// TIA Portal V17 export
// export: Created 2023-02-25T15:48:13.2517899Z, ExportSetting WithDefaults, DisplayName Totally Integrated Automation Portal, DisplayVersion V17, DisplayName TIA Portal Openness, DisplayVersion V17, DisplayName TIA Portal Version Control Interface, DisplayVersion V17, DisplayName TIA Portal Test Suite Advanced, DisplayVersion V17, DisplayName STEP 7 Professional, DisplayVersion V17, DisplayName SIMATIC Energy Suite, DisplayVersion V17, DisplayName STEP 7 Safety, DisplayVersion V17, DisplayName WinCC Professional, DisplayVersion V17
FUNCTION_BLOCK "LOG_AutoControle"   // FB5, LAD
TITLE = Auto Controle - Sequential algorithm
{ S7_Optimized_Access := 'TRUE' }
VERSION : 0.1
// stored: AutoNumber true, IsIECCheckEnabled false, IsRetainMemResEnabled false, MemoryReserve 100, SetENOAutomatically false, UDAEnableTagReadback false
   VAR_INPUT
      StartLine : Bool;
      StopLine : Bool;
      AutoMode : Bool;
      SmallPackage : Bool;
      MediumPackage : Bool;
      LargePackage : Bool;
      D3 : Bool;
      D4 : Bool;
      D5 : Bool;
      D6 : Bool;
      FirstScan : Bool;
   END_VAR
   VAR_OUTPUT
      ConveyorsAuto : "stt_Conveyor";
   END_VAR
   VAR
      s1 : Bool;
      s2 : Bool;
      s3 : Bool;
      s4 : Bool;
      s5 : Bool;
      P_D3_1 : Bool;
      P_D3_2 : Bool;
      P_D3_3 : Bool;
      N_D4 : Bool;
      N_D5 : Bool;
      N_D6 : Bool;
   END_VAR
   VAR_TEMP   // added for the SCL form of the ladder/FBD networks
      _w1 : Bool;
   END_VAR
BEGIN

REGION Network 1: Step 3-2
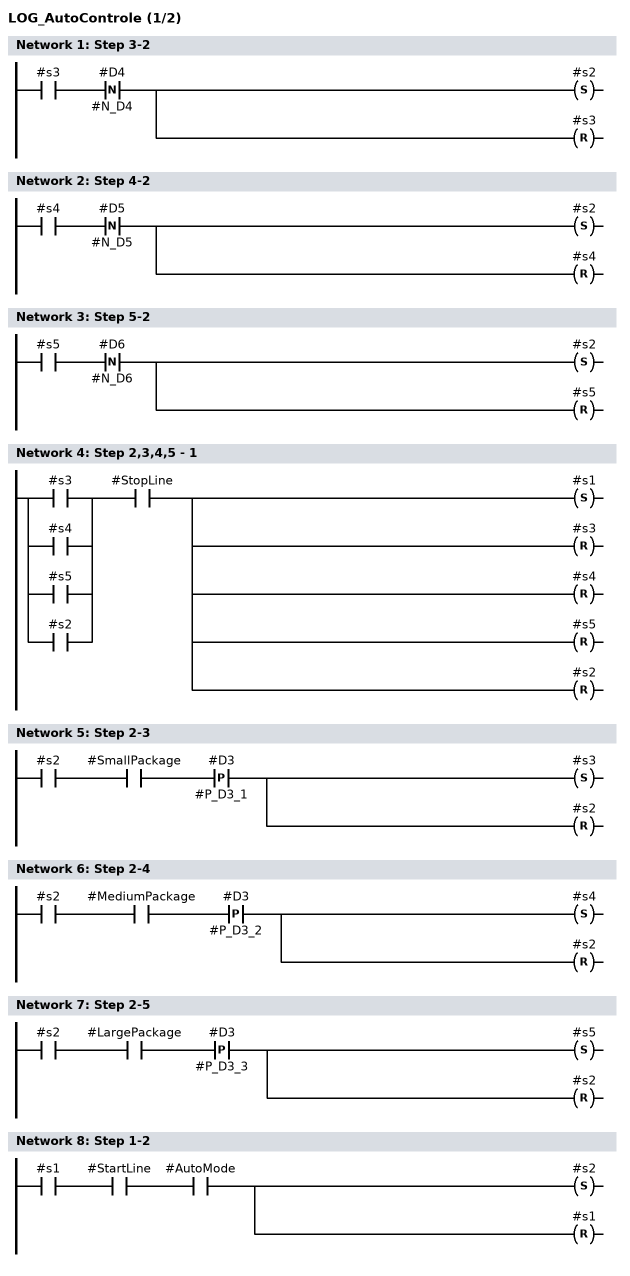
   RUNG wire#powerrail
      Contact( #s3 )
      N_Contact(operand := #D4, bit := #N_D4)
      wire#w1
      S_Coil( #s2 )
   END_RUNG
   RUNG wire#w1
      R_Coil( #s3 )
   END_RUNG
   // the same network as SCL:
   #_w1 := #s3 AND NOT #D4 AND #N_D4;   // falling edge of #D4
   #N_D4 := #D4;
   IF #_w1 THEN
       #s2 := TRUE;
       #s3 := FALSE;
   END_IF;
END_REGION

REGION Network 2: Step 4-2
   RUNG wire#powerrail
      Contact( #s4 )
      N_Contact(operand := #D5, bit := #N_D5)
      wire#w1
      S_Coil( #s2 )
   END_RUNG
   RUNG wire#w1
      R_Coil( #s4 )
   END_RUNG
   // the same network as SCL:
   #_w1 := #s4 AND NOT #D5 AND #N_D5;   // falling edge of #D5
   #N_D5 := #D5;
   IF #_w1 THEN
       #s2 := TRUE;
       #s4 := FALSE;
   END_IF;
END_REGION

REGION Network 3: Step 5-2
   RUNG wire#powerrail
      Contact( #s5 )
      N_Contact(operand := #D6, bit := #N_D6)
      wire#w1
      S_Coil( #s2 )
   END_RUNG
   RUNG wire#w1
      R_Coil( #s5 )
   END_RUNG
   // the same network as SCL:
   #_w1 := #s5 AND NOT #D6 AND #N_D6;   // falling edge of #D6
   #N_D6 := #D6;
   IF #_w1 THEN
       #s2 := TRUE;
       #s5 := FALSE;
   END_IF;
END_REGION

REGION Network 4: Step 2,3,4,5 - 1
   RUNG wire#powerrail
      Contact( #s3 )
      wire#w1
      Contact( #StopLine )
      wire#w2
      S_Coil( #s1 )
   END_RUNG
   RUNG wire#powerrail
      Contact( #s4 )
   END_RUNG wire#w1
   RUNG wire#powerrail
      Contact( #s5 )
   END_RUNG wire#w1
   RUNG wire#powerrail
      Contact( #s2 )
   END_RUNG wire#w1
   RUNG wire#w2
      R_Coil( #s3 )
   END_RUNG
   RUNG wire#w2
      R_Coil( #s4 )
   END_RUNG
   RUNG wire#w2
      R_Coil( #s5 )
   END_RUNG
   RUNG wire#w2
      R_Coil( #s2 )
   END_RUNG
   // the same network as SCL:
   IF (#s3 OR #s4 OR #s5 OR #s2) AND #StopLine THEN #s1 := TRUE; END_IF;
   #_w1 := (#s3 OR #s4 OR #s5 OR #s2) AND #StopLine;
   IF #_w1 THEN
       #s3 := FALSE;
       #s4 := FALSE;
       #s5 := FALSE;
       #s2 := FALSE;
   END_IF;
END_REGION

REGION Network 5: Step 2-3
   RUNG wire#powerrail
      Contact( #s2 )
      Contact( #SmallPackage )
      P_Contact(operand := #D3, bit := #P_D3_1)
      wire#w1
      S_Coil( #s3 )
   END_RUNG
   RUNG wire#w1
      R_Coil( #s2 )
   END_RUNG
   // the same network as SCL:
   #_w1 := #s2 AND #SmallPackage AND #D3 AND NOT #P_D3_1;   // rising edge of #D3
   #P_D3_1 := #D3;
   IF #_w1 THEN
       #s3 := TRUE;
       #s2 := FALSE;
   END_IF;
END_REGION

REGION Network 6: Step 2-4
   RUNG wire#powerrail
      Contact( #s2 )
      Contact( #MediumPackage )
      P_Contact(operand := #D3, bit := #P_D3_2)
      wire#w1
      S_Coil( #s4 )
   END_RUNG
   RUNG wire#w1
      R_Coil( #s2 )
   END_RUNG
   // the same network as SCL:
   #_w1 := #s2 AND #MediumPackage AND #D3 AND NOT #P_D3_2;   // rising edge of #D3
   #P_D3_2 := #D3;
   IF #_w1 THEN
       #s4 := TRUE;
       #s2 := FALSE;
   END_IF;
END_REGION

REGION Network 7: Step 2-5
   RUNG wire#powerrail
      Contact( #s2 )
      Contact( #LargePackage )
      P_Contact(operand := #D3, bit := #P_D3_3)
      wire#w1
      S_Coil( #s5 )
   END_RUNG
   RUNG wire#w1
      R_Coil( #s2 )
   END_RUNG
   // the same network as SCL:
   #_w1 := #s2 AND #LargePackage AND #D3 AND NOT #P_D3_3;   // rising edge of #D3
   #P_D3_3 := #D3;
   IF #_w1 THEN
       #s5 := TRUE;
       #s2 := FALSE;
   END_IF;
END_REGION

REGION Network 8: Step 1-2
   RUNG wire#powerrail
      Contact( #s1 )
      Contact( #StartLine )
      Contact( #AutoMode )
      wire#w1
      S_Coil( #s2 )
   END_RUNG
   RUNG wire#w1
      R_Coil( #s1 )
   END_RUNG
   // the same network as SCL:
   IF #s1 AND #StartLine AND #AutoMode THEN
       #s2 := TRUE;
       #s1 := FALSE;
   END_IF;
END_REGION

REGION Network 9: Step 2,3,4,5 Output
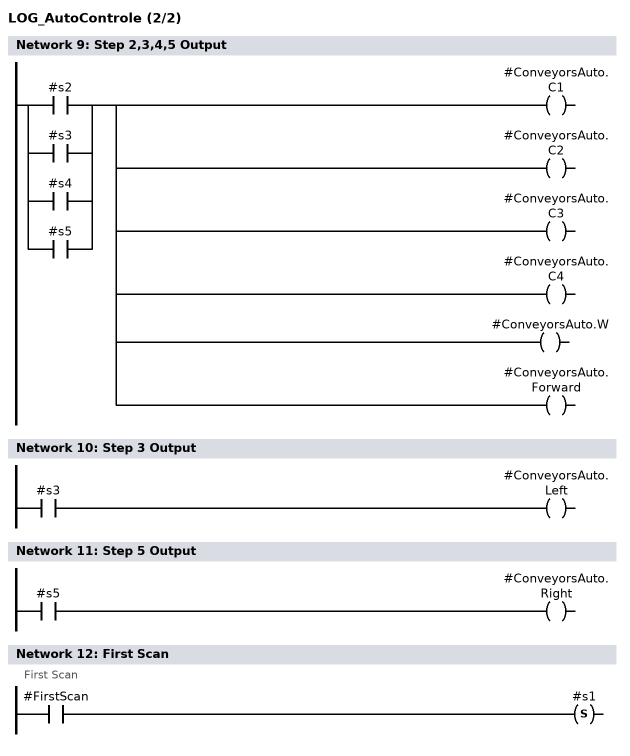
   RUNG wire#powerrail
      Contact( #s2 )
      wire#w1
      Coil( #ConveyorsAuto.C1 )
   END_RUNG
   RUNG wire#powerrail
      Contact( #s3 )
   END_RUNG wire#w1
   RUNG wire#powerrail
      Contact( #s4 )
   END_RUNG wire#w1
   RUNG wire#powerrail
      Contact( #s5 )
   END_RUNG wire#w1
   RUNG wire#w1
      Coil( #ConveyorsAuto.C2 )
   END_RUNG
   RUNG wire#w1
      Coil( #ConveyorsAuto.C3 )
   END_RUNG
   RUNG wire#w1
      Coil( #ConveyorsAuto.C4 )
   END_RUNG
   RUNG wire#w1
      Coil( #ConveyorsAuto.W )
   END_RUNG
   RUNG wire#w1
      Coil( #ConveyorsAuto.Forward )
   END_RUNG
   // the same network as SCL:
   #ConveyorsAuto.C1 := #s2 OR #s3 OR #s4 OR #s5;
   #ConveyorsAuto.C2 := #ConveyorsAuto.C1;
   #ConveyorsAuto.C3 := #ConveyorsAuto.C1;
   #ConveyorsAuto.C4 := #ConveyorsAuto.C1;
   #ConveyorsAuto.W := #ConveyorsAuto.C1;
   #ConveyorsAuto.Forward := #ConveyorsAuto.C1;
END_REGION

REGION Network 10: Step 3 Output
   RUNG wire#powerrail
      Contact( #s3 )
      Coil( #ConveyorsAuto.Left )
   END_RUNG
   // the same network as SCL:
   #ConveyorsAuto.Left := #s3;
END_REGION

REGION Network 11: Step 5 Output
   RUNG wire#powerrail
      Contact( #s5 )
      Coil( #ConveyorsAuto.Right )
   END_RUNG
   // the same network as SCL:
   #ConveyorsAuto.Right := #s5;
END_REGION

REGION Network 12: First Scan
   // First Scan
   RUNG wire#powerrail
      Contact( #FirstScan )
      S_Coil( #s1 )
   END_RUNG
   // the same network as SCL:
   IF #FirstScan THEN #s1 := TRUE; END_IF;
END_REGION
END_FUNCTION_BLOCK
